SMOVL C00398 BC00398 V=800.0  +MOVJ EC00398
SMOVL C00399 BC00399 V=1000.0  +MOVJ EC00399
SMOVL C00400 BC00400 V=1000.0  +MOVJ EC00400
SFTOF3D
'EndPath W3863
MOVJ C00401 BC00401 VJ=100.00  +MOVJ EC00401 VJ=100.00
MOVJ C00402 BC00402 VJ=100.00  +MOVJ EC00402 VJ=100.00
'Path W3864
SFTOF3D
SFTON3D P033
MOVJ C00403 BC00403 VJ=100.00  +MOVJ EC00403 VJ=100.00
SMOVL C00404 BC00404 V=800.0  +MOVJ EC00404
SMOVL C00405 BC00405 V=166.7 PL=0  +MOVJ EC00405
ARCON
SMOVL C00406 BC00406 V=10.0  +MOVJ EC00406
SFTON3D P034
SMOVL C00407 BC00407 V=10.0  +MOVJ EC00407
SMOVL C00408 BC00408 V=10.0  +MOVJ EC00408
ARCOF
SMOVL C00409 BC00409 V=800.0  +MOVJ EC00409
SMOVL C00410 BC00410 V=1000.0  +MOVJ EC00410
SMOVL C00411 BC00411 V=1000.0  +MOVJ EC00411
SFTOF3D
'EndPath W3864
MOVJ C00412 BC00412 VJ=100.00  +MOVJ EC00412 VJ=100.00
'Path W3865
SFTOF3D
SFTON3D P032
MOVJ C00413 BC00413 VJ=100.00  +MOVJ EC00413 VJ=100.00
MOVJ C00414 BC00414 VJ=100.00  +MOVJ EC00414 VJ=100.00
SMOVL C00415 BC00415 V=800.0  +MOVJ EC00415
SMOVL C00416 BC00416 V=166.7 PL=0  +MOVJ EC00416
ARCON
SMOVL C00417 BC00417 V=9.2  +MOVJ EC00417
SFTON3D P031
SMOVL C00418 BC00418 V=9.2  +MOVJ EC00418
SMOVL C00419 BC00419 V=9.2  +MOVJ EC00419
ARCOF
SMOVL C00420 BC00420 V=800.0  +MOVJ EC00420
SMOVL C00421 BC00421 V=1000.0  +MOVJ EC00421
SFTOF3D
'EndPath W3865
MOVJ C00422 BC00422 VJ=100.00  +MOVJ EC00422 VJ=100.00
'Down
MOVJ C00423 BC00423 VJ=100.00  +MOVJ EC00423 VJ=100.00
MOVJ C00424 BC00424 VJ=100.00  +MOVJ EC00424 VJ=100.00
'Path W3867
SFTOF3D
SFTON3D P026
MOVJ C00425 BC00425 VJ=100.00  +MOVJ EC00425 VJ=100.00
SMOVL C00426 BC00426 V=800.0  +MOVJ EC00426
SMOVL C00427 BC00427 V=150.0 PL=0  +MOVJ EC00427
MACRO1 MJ#(0) ARGF22
ARCON
SMOVC C00428 BC00428 V=9.5  +MOVJ EC00428
SMOVC C00429 BC00429 V=9.5  +MOVJ EC00429
SFTON3D P025
SMOVC C00430 BC00430 V=9.5  +MOVJ EC00430
SMOVL C00431 BC00431 V=9.5  +MOVJ EC00431
ARCOF
SMOVL C00432 BC00432 V=800.0  +MOVJ EC00432
SMOVL C00433 BC00433 V=1000.0  +MOVJ EC00433
SFTOF3D
'EndPath W3867
MOVJ C00434 BC00434 VJ=100.00  +MOVJ EC00434 VJ=100.00
MOVJ C00435 BC00435 VJ=100.00  +MOVJ EC00435 VJ=100.00
MOVJ C00436 BC00436 VJ=100.00  +MOVJ EC00436 VJ=100.00
'Path W3868
SFTOF3D
SFTON3D P022
MOVJ C00437 BC00437 VJ=100.00  +MOVJ EC00437 VJ=100.00
MOVJ C00438 BC00438 VJ=100.00  +MOVJ EC00438 VJ=100.00
SMOVL C00439 BC00439 V=800.0  +MOVJ EC00439
SMOVL C00440 BC00440 V=166.7 PL=0  +MOVJ EC00440
MACRO1 MJ#(0) ARGF9
ARCON
SMOVL C00441 BC00441 V=10.0  +MOVJ EC00441
SMOVL C00442 BC00442 V=10.0  +MOVJ EC00442
SMOVL C00443 BC00443 V=10.0  +MOVJ EC00443
SMOVL C00444 BC00444 V=10.0  +MOVJ EC00444
SMOVL C00445 BC00445 V=10.0  +MOVJ EC00445
SMOVL C00446 BC00446 V=10.0  +MOVJ EC00446
SMOVL C00447 BC00447 V=10.0  +MOVJ EC00447
SMOVL C00448 BC00448 V=10.0  +MOVJ EC00448
SMOVL C00449 BC00449 V=10.0  +MOVJ EC00449
ARCOF
SMOVL C00450 BC00450 V=800.0  +MOVJ EC00450
SMOVL C00451 BC00451 V=1000.0  +MOVJ EC00451
SFTOF3D
'EndPath W3868
MOVJ C00452 BC00452 VJ=100.00  +MOVJ EC00452 VJ=100.00
SFTOF3D
'EndPath W3869
MOVJ C00453 BC00453 VJ=100.00  +MOVJ EC00453 VJ=100.00
'Path W3896
SFTOF3D
SFTON3D P020
MOVJ C00454 BC00454 VJ=100.00  +MOVJ EC00454 VJ=100.00
SMOVL C00455 BC00455 V=800.0  +MOVJ EC00455
SMOVL C00456 BC00456 V=150.0 PL=0  +MOVJ EC00456
ARCON
SMOVL C00457 BC00457 V=10.0  +MOVJ EC00457
ARCOF
SMOVL C00458 BC00458 V=800.0  +MOVJ EC00458
SFTOF3D
'EndPath W3896
MOVJ C00459 BC00459 VJ=100.00  +MOVJ EC00459 VJ=100.00
MOVJ C00460 BC00460 VJ=100.00  +MOVJ EC00460 VJ=100.00
MOVJ C00461 BC00461 VJ=100.00  +MOVJ EC00461 VJ=100.00
'Path W3866
SFTOF3D
SFTON3D P023
MOVJ C00462 BC00462 VJ=100.00  +MOVJ EC00462 VJ=100.00
SMOVL C00463 BC00463 V=800.0  +MOVJ EC00463
SMOVC C00464 BC00464 V=150.0 PL=0  +MOVJ EC00464
MACRO1 MJ#(0) ARGF22
ARCON
SWVON WEV#(108)
SMOVC C00465 BC00465 V=9.5  +MOVJ EC00465
SMOVC C00466 BC00466 V=9.5  +MOVJ EC00466
SFTON3D P024
SMOVC C00467 BC00467 V=9.5  +MOVJ EC00467
SMOVC C00468 BC00468 V=9.5  +MOVJ EC00468
SMOVC C00469 BC00469 V=9.5  +MOVJ EC00469
ARCOF
SWVOF
SMOVL C00470 BC00470 V=800.0  +MOVJ EC00470
SMOVL C00471 BC00471 V=1000.0  +MOVJ EC00471
SFTOF3D
'EndPath W3866
MOVJ C00472 BC00472 VJ=100.00  +MOVJ EC00472 VJ=100.00
MOVJ C00473 BC00473 VJ=100.00  +MOVJ EC00473 VJ=100.00
SFTOF3D
MOVJ C00474 BC00474 VJ=100.00  +MOVJ EC00474 VJ=100.00
SMOVL C00475 BC00475 V=800.0  +MOVJ EC00475
MOVJ C00476 BC00476 VJ=100.00  +MOVJ EC00476 VJ=100.00
SFTON3D P056
MOVJ C00477 BC00477 VJ=100.00  +MOVJ EC00477 VJ=100.00
SMOVL C00478 BC00478 V=150.0 PL=0  +MOVJ EC00478
MACRO1 MJ#(0) ARGF9
ARCON
SFTON3D P057
SMOVL C00479 BC00479 V=10.0  +MOVJ EC00479
SMOVC C00480 BC00480 V=13.3  +MOVJ EC00480
SMOVC C00481 BC00481 V=13.3  +MOVJ EC00481
SMOVC C00482 BC00482 V=13.3  +MOVJ EC00482
SFTON3D P056
SMOVL C00483 BC00483 V=10.0  +MOVJ EC00483
SMOVL C00484 BC00484 V=10.0  +MOVJ EC00484
SMOVC C00485 BC00485 V=13.3  +MOVJ EC00485
SMOVC C00486 BC00486 V=13.3  +MOVJ EC00486
SMOVC C00487 BC00487 V=13.3  +MOVJ EC00487
ARCOF
SMOVL C00488 BC00488 V=166.7  +MOVJ EC00488
SFTOF3D
SMOVL C00489 BC00489 V=666.7  +MOVJ EC00489
SMOVL C00490 BC00490 V=666.7  +MOVJ EC00490
SFTON3D P054
SMOVL C00491 BC00491 V=150.0 PL=0  +MOVJ EC00491
MACRO1 MJ#(0) ARGF9
ARCON
SFTON3D P055
SMOVL C00492 BC00492 V=10.0  +MOVJ EC00492
SMOVC C00493 BC00493 V=13.3  +MOVJ EC00493
SMOVC C00494 BC00494 V=13.3  +MOVJ EC00494
SMOVC C00495 BC00495 V=13.3  +MOVJ EC00495
SFTON3D P054
SMOVL C00496 BC00496 V=10.0  +MOVJ EC00496
SMOVL C00497 BC00497 V=10.0  +MOVJ EC00497
SMOVC C00498 BC00498 V=13.3  +MOVJ EC00498
SMOVC C00499 BC00499 V=13.3  +MOVJ EC00499
SMOVC C00500 BC00500 V=13.3  +MOVJ EC00500
ARCOF
SMOVL C00501 BC00501 V=166.7  +MOVJ EC00501
SFTOF3D
MOVL C00502 BC00502 V=666.7  +MOVJ EC00502 VJ=0.78
MOVL C00503 BC00503 V=666.7  +MOVJ EC00503 VJ=0.78
MOVL C00504 BC00504 V=666.7  +MOVJ EC00504 VJ=0.78
MOVJ C00505 BC00505 VJ=100.00  +MOVJ EC00505 VJ=0.78
SFTON3D P060
SMOVL C00506 BC00506 V=150.0 PL=0  +MOVJ EC00506
MACRO1 MJ#(0) ARGF9
ARCON
SFTON3D P061
SMOVL C00507 BC00507 V=10.0  +MOVJ EC00507
SMOVC C00508 BC00508 V=15.0  +MOVJ EC00508
SMOVC C00509 BC00509 V=15.0  +MOVJ EC00509
SMOVC C00510 BC00510 V=13.3  +MOVJ EC00510
SFTON3D P060
SMOVL C00511 BC00511 V=10.0  +MOVJ EC00511
SMOVL C00512 BC00512 V=10.0  +MOVJ EC00512
SMOVC C00513 BC00513 V=13.3  +MOVJ EC00513
SMOVC C00514 BC00514 V=13.3  +MOVJ EC00514
SMOVC C00515 BC00515 V=15.0  +MOVJ EC00515
ARCOF
SMOVL C00516 BC00516 V=166.7  +MOVJ EC00516
SFTOF3D
MOVJ C00517 BC00517 VJ=100.00  +MOVJ EC00517 VJ=100.00
MOVJ C00518 BC00518 VJ=100.00  +MOVJ EC00518 VJ=100.00
SFTON3D P059
SMOVL C00519 BC00519 V=150.0 PL=0  +MOVJ EC00519
MACRO1 MJ#(0) ARGF9
ARCON
SFTON3D P058
SMOVL C00520 BC00520 V=10.0  +MOVJ EC00520
SMOVC C00521 BC00521 V=13.3  +MOVJ EC00521
SMOVC C00522 BC00522 V=13.3  +MOVJ EC00522
SMOVC C00523 BC00523 V=13.3  +MOVJ EC00523
SFTON3D P059
SMOVL C00524 BC00524 V=10.0  +MOVJ EC00524
SMOVL C00525 BC00525 V=10.0  +MOVJ EC00525
SMOVC C00526 BC00526 V=13.3  +MOVJ EC00526
SMOVC C00527 BC00527 V=13.3  +MOVJ EC00527
SMOVC C00528 BC00528 V=13.3  +MOVJ EC00528
ARCOF
SMOVL C00529 BC00529 V=166.7  +MOVJ EC00529
SFTOF3D
MOVJ C00530 BC00530 VJ=100.00  +MOVJ EC00530 VJ=100.00
MOVJ C00531 BC00531 VJ=100.00  +MOVJ EC00531 VJ=100.00
SFTON3D P063
SMOVL C00532 BC00532 V=150.0 PL=0  +MOVJ EC00532
MACRO1 MJ#(0) ARGF9
ARCON
SFTON3D P062
SMOVL C00533 BC00533 V=10.0  +MOVJ EC00533
SMOVC C00534 BC00534 V=13.3  +MOVJ EC00534
SMOVC C00535 BC00535 V=13.3  +MOVJ EC00535
SMOVC C00536 BC00536 V=13.3  +MOVJ EC00536
SFTON3D P063
SMOVL C00537 BC00537 V=10.0  +MOVJ EC00537
SMOVL C00538 BC00538 V=10.0  +MOVJ EC00538
SMOVC C00539 BC00539 V=13.3  +MOVJ EC00539
SMOVC C00540 BC00540 V=13.3  +MOVJ EC00540
SMOVC C00541 BC00541 V=13.3  +MOVJ EC00541
ARCOF
SMOVL C00542 BC00542 V=166.7  +MOVJ EC00542
SFTOF3D
MOVJ C00543 BC00543 VJ=100.00  +MOVJ EC00543 VJ=100.00
MOVJ C00544 BC00544 VJ=100.00  +MOVJ EC00544 VJ=100.00
SFTON3D P072
SMOVL C00545 BC00545 V=150.0 PL=0  +MOVJ EC00545
MACRO1 MJ#(0) ARGF9
ARCON
SFTON3D P071
SMOVL C00546 BC00546 V=10.0  +MOVJ EC00546
SMOVC C00547 BC00547 V=13.3  +MOVJ EC00547
SMOVC C00548 BC00548 V=13.3  +MOVJ EC00548
SMOVC C00549 BC00549 V=13.3  +MOVJ EC00549
SMOVL C00550 BC00550 V=10.0  +MOVJ EC00550
SFTON3D P070
SMOVL C00551 BC00551 V=10.0  +MOVJ EC00551
SMOVL C00552 BC00552 V=10.0  +MOVJ EC00552
ARCOF
SMOVL C00553 BC00553 V=166.7  +MOVJ EC00553
SFTOF3D
MOVJ C00554 BC00554 VJ=100.00  +MOVJ EC00554 VJ=100.00
MOVJ C00555 BC00555 VJ=100.00  +MOVJ EC00555 VJ=100.00
SFTON3D P065
SMOVL C00556 BC00556 V=150.0 PL=0  +MOVJ EC00556
MACRO1 MJ#(0) ARGF9
ARCON
SFTON3D P064
SMOVL C00557 BC00557 V=10.0  +MOVJ EC00557
SMOVC C00558 BC00558 V=13.3  +MOVJ EC00558
SMOVC C00559 BC00559 V=13.3  +MOVJ EC00559
SMOVC C00560 BC00560 V=13.3  +MOVJ EC00560
SFTON3D P065
SMOVL C00561 BC00561 V=10.0  +MOVJ EC00561
SMOVL C00562 BC00562 V=10.0  +MOVJ EC00562
SMOVC C00563 BC00563 V=13.3  +MOVJ EC00563
SMOVC C00564 BC00564 V=13.3  +MOVJ EC00564
SMOVC C00565 BC00565 V=13.3  +MOVJ EC00565
ARCOF
SMOVL C00566 BC00566 V=166.7  +MOVJ EC00566
SFTOF3D
MOVJ C00567 BC00567 VJ=100.00  +MOVJ EC00567 VJ=100.00
MOVJ C00568 BC00568 VJ=100.00  +MOVJ EC00568 VJ=100.00
MOVJ C00569 BC00569 VJ=100.00  +MOVJ EC00569 VJ=100.00
SFTON3D P051
SMOVL C00570 BC00570 V=150.0 PL=0  +MOVJ EC00570
MACRO1 MJ#(0) ARGF9
ARCON
SMOVL C00571 BC00571 V=10.8  +MOVJ EC00571
SMOVC C00572 BC00572 V=13.3  +MOVJ EC00572
SMOVC C00573 BC00573 V=13.3  +MOVJ EC00573
SMOVC C00574 BC00574 V=13.3  +MOVJ EC00574
SFTON3D P052
SMOVL C00575 BC00575 V=11.7  +MOVJ EC00575
SFTON3D P053
SMOVL C00576 BC00576 V=11.7  +MOVJ EC00576
SMOVC C00577 BC00577 V=13.3  +MOVJ EC00577
SMOVC C00578 BC00578 V=13.3  +MOVJ EC00578
SMOVC C00579 BC00579 V=13.3  +MOVJ EC00579
ARCOF
SMOVL C00580 BC00580 V=166.7  +MOVJ EC00580
SFTOF3D
MOVL C00581 BC00581 V=1000.0  +MOVJ EC00581 VJ=100.00
MOVJ C00582 BC00582 VJ=100.00  +MOVJ EC00582 VJ=100.00
CALL JOB:CLEAN-R1_KM_3P
MOVJ C00583 BC00583 VJ=100.00  +MOVJ EC00583 VJ=0.78
MOVJ C00584 BC00584 VJ=100.00  +MOVJ EC00584 VJ=100.00
MOVJ C00585 BC00585 VJ=100.00  +MOVJ EC00585 VJ=100.00
MOVJ C00586 BC00586 VJ=100.00  +MOVJ EC00586 VJ=100.00
MOVJ C00587 BC00587 VJ=100.00  +MOVJ EC00587 VJ=100.00
MOVJ C00588 BC00588 VJ=100.00  +MOVJ EC00588 VJ=100.00
MOVJ C00589 BC00589 VJ=100.00  +MOVJ EC00589 VJ=100.00
MOVJ C00590 BC00590 VJ=100.00  +MOVJ EC00590 VJ=100.00
MOVJ C00591 BC00591 VJ=100.00  +MOVJ EC00591 VJ=100.00
MOVJ C00592 BC00592 VJ=100.00  +MOVJ EC00592 VJ=100.00
SMOVL C00593 BC00593 V=333.3  +MOVJ EC00593
SMOVL C00594 BC00594 V=333.3  +MOVJ EC00594
MOVJ C00595 BC00595 VJ=100.00  +MOVJ EC00595 VJ=100.00
SMOVL C00596 BC00596 V=333.3  +MOVJ EC00596
SMOVL C00597 BC00597 V=166.7  +MOVJ EC00597
SREFP 3 C00598 BC00598  +REFP EC00598
CALL JOB:SEARCH-R1-S13D
SET P051 P006
SFTON3D P051
SMOVL C00599 BC00599 V=166.7  +MOVJ EC00599
SREFP 3 C00600 BC00600  +REFP EC00600
CALL JOB:SEARCH-R1-S13D
SET P051 P006
SFTON3D P051
SMOVL C00601 BC00601 V=166.7  +MOVJ EC00601
SREFP 3 C00602 BC00602  +REFP EC00602
CALL JOB:SEARCH-R1-S13D
SET P051 P006
SFTON3D P051
SMOVL C00603 BC00603 V=166.7  +MOVJ EC00603
SMOVL C00604 BC00604 V=166.7 PL=0  +MOVJ EC00604
SMOVL C00605 BC00605 V=166.7  +MOVJ EC00605
SREFP 3 C00606 BC00606  +REFP EC00606
CALL JOB:SEARCH-R1-S13D
SET P052 P006
SFTON3D P052
SMOVL C00607 BC00607 V=166.7  +MOVJ EC00607
SREFP 3 C00608 BC00608  +REFP EC00608
CALL JOB:SEARCH-R1-S13D
SET P052 P006
SFTON3D P052
SMOVL C00609 BC00609 V=166.7  +MOVJ EC00609
SMOVL C00610 BC00610 V=333.3 PL=0  +MOVJ EC00610
SMOVL C00611 BC00611 V=166.7  +MOVJ EC00611
SREFP 3 C00612 BC00612  +REFP EC00612
CALL JOB:SEARCH-R1-S13D
SET P053 P006
SFTON3D P053
SMOVL C00613 BC00613 V=166.7  +MOVJ EC00613
SREFP 3 C00614 BC00614  +REFP EC00614
CALL JOB:SEARCH-R1-S13D
SET P053 P006
SFTON3D P053
SMOVL C00615 BC00615 V=166.7  +MOVJ EC00615
SFTOF3D
SFTOF
SFTON3D P051
SMOVL C00616 BC00616 V=333.3  +MOVJ EC00616
SMOVL C00617 BC00617 V=166.7  +MOVJ EC00617
SREFP 3 C00618 BC00618  +REFP EC00618
CALL JOB:SEARCH-R1-S13D
SET P050 P006
SFTON3D P050
SMOVL C00619 BC00619 V=166.7  +MOVJ EC00619
SREFP 3 C00620 BC00620  +REFP EC00620
CALL JOB:SEARCH-R1-S13D
SET P050 P006
SFTON3D P050
SMOVL C00621 BC00621 V=166.7  +MOVJ EC00621
SMOVL C00622 BC00622 V=166.7  +MOVJ EC00622
SREFP 3 C00623 BC00623  +REFP EC00623
CALL JOB:SEARCH-R1-S13D
SET P050 P006
SFTON3D P050
SMOVL C00624 BC00624 V=166.7  +MOVJ EC00624
SFTOF3D
SMOVL C00625 BC00625 V=333.3  +MOVJ EC00625
SMOVL C00626 BC00626 V=166.7  +MOVJ EC00626
SREFP 3 C00627 BC00627  +REFP EC00627
CALL JOB:SEARCH-R1-S13D
SET P054 P006
SFTON3D P054
SMOVL C00628 BC00628 V=166.7  +MOVJ EC00628
SREFP 3 C00629 BC00629  +REFP EC00629
CALL JOB:SEARCH-R1-S13D
SET P054 P006
SFTON3D P054
SMOVL C00630 BC00630 V=166.7  +MOVJ EC00630
SMOVL C00631 BC00631 V=166.7  +MOVJ EC00631
SREFP 3 C00632 BC00632  +REFP EC00632
CALL JOB:SEARCH-R1-S13D
SET P054 P006
SFTON3D P054
SMOVL C00633 BC00633 V=166.7  +MOVJ EC00633
SMOVL C00634 BC00634 V=333.3  +MOVJ EC00634
SMOVL C00635 BC00635 V=166.7  +MOVJ EC00635
SREFP 3 C00636 BC00636  +REFP EC00636
CALL JOB:SEARCH-R1-S13D
SET P055 P006
SFTON3D P055
SMOVL C00637 BC00637 V=166.7  +MOVJ EC00637
SREFP 3 C00638 BC00638  +REFP EC00638
CALL JOB:SEARCH-R1-S13D
SET P055 P006
SFTON3D P055
SMOVL C00639 BC00639 V=166.7  +MOVJ EC00639
SREFP 3 C00640 BC00640  +REFP EC00640
CALL JOB:SEARCH-R1-S13D
SET P055 P006
SFTON3D P055
SMOVL C00641 BC00641 V=166.7  +MOVJ EC00641
MOVJ C00642 BC00642 VJ=100.00  +MOVJ EC00642 VJ=100.00
MOVL C00643 BC00643 V=333.3  +MOVJ EC00643 VJ=100.00
SMOVL C00644 BC00644 V=166.7  +MOVJ EC00644
SREFP 3 C00645 BC00645  +REFP EC00645
CALL JOB:SEARCH-R1-S13D
SET P056 P006
SFTON3D P056
SMOVL C00646 BC00646 V=166.7  +MOVJ EC00646
SREFP 3 C00647 BC00647  +REFP EC00647
CALL JOB:SEARCH-R1-S13D
SET P056 P006
SFTON3D P056
SMOVL C00648 BC00648 V=166.7  +MOVJ EC00648
SMOVL C00649 BC00649 V=333.3  +MOVJ EC00649
SMOVL C00650 BC00650 V=166.7  +MOVJ EC00650
SREFP 3 C00651 BC00651  +REFP EC00651
CALL JOB:SEARCH-R1-S13D
SET P057 P006
SFTON3D P057
SMOVL C00652 BC00652 V=166.7  +MOVJ EC00652
SREFP 3 C00653 BC00653  +REFP EC00653
CALL JOB:SEARCH-R1-S13D
SET P057 P006
SFTON3D P057
SMOVL C00654 BC00654 V=166.7  +MOVJ EC00654
SMOVL C00655 BC00655 V=333.3  +MOVJ EC00655
SMOVL C00656 BC00656 V=166.7  +MOVJ EC00656
SREFP 3 C00657 BC00657  +REFP EC00657
CALL JOB:SEARCH-R1-S13D
SET P058 P006
SFTON3D P058
SMOVL C00658 BC00658 V=166.7  +MOVJ EC00658
SREFP 3 C00659 BC00659  +REFP EC00659
CALL JOB:SEARCH-R1-S13D
SET P058 P006
SFTON3D P058
SMOVL C00660 BC00660 V=166.7  +MOVJ EC00660
SFTOF3D
MOVL C00661 BC00661 V=333.3  +MOVJ EC00661 VJ=100.00
MOVL C00662 BC00662 V=333.3  +MOVJ EC00662 VJ=100.00
SMOVL C00663 BC00663 V=166.7  +MOVJ EC00663
SREFP 3 C00664 BC00664  +REFP EC00664
CALL JOB:SEARCH-R1-S13D
SET P059 P006
SFTON3D P059
SMOVL C00665 BC00665 V=166.7  +MOVJ EC00665
SREFP 3 C00666 BC00666  +REFP EC00666
CALL JOB:SEARCH-R1-S13D
SET P059 P006
SFTON3D P059
SMOVL C00667 BC00667 V=166.7  +MOVJ EC00667
SREFP 3 C00668 BC00668  +REFP EC00668
CALL JOB:SEARCH-R1-S13D
SET P059 P006
SFTON3D P059
SMOVL C00669 BC00669 V=166.7  +MOVJ EC00669
MOVL C00670 BC00670 V=333.3  +MOVJ EC00670 VJ=100.00
SMOVL C00671 BC00671 V=166.7  +MOVJ EC00671
SREFP 3 C00672 BC00672  +REFP EC00672
CALL JOB:SEARCH-R1-S13D
SET P060 P006
SFTON3D P060
SMOVL C00673 BC00673 V=166.7  +MOVJ EC00673
SREFP 3 C00674 BC00674  +REFP EC00674
CALL JOB:SEARCH-R1-S13D
SET P060 P006
SFTON3D P060
SMOVL C00675 BC00675 V=166.7  +MOVJ EC00675
SREFP 3 C00676 BC00676  +REFP EC00676
CALL JOB:SEARCH-R1-S13D
SET P060 P006
SFTON3D P060
SMOVL C00677 BC00677 V=166.7  +MOVJ EC00677
SFTOF3D
SFTON3D P060
MACRO1 MJ#(0) ARGF9
SMOVL C00678 BC00678 V=150.0 PL=0  +MOVJ EC00678
ARCON
SMOVL C00679 BC00679 V=10.0  +MOVJ EC00679
SMOVC C00680 BC00680 V=13.3  +MOVJ EC00680
SMOVC C00681 BC00681 V=13.3  +MOVJ EC00681
SMOVC C00682 BC00682 V=13.3  +MOVJ EC00682
SFTON3D P059
SMOVL C00683 BC00683 V=10.0  +MOVJ EC00683
SMOVL C00684 BC00684 V=10.0  +MOVJ EC00684
SMOVC C00685 BC00685 V=13.3  +MOVJ EC00685
SMOVC C00686 BC00686 V=13.3  +MOVJ EC00686
SMOVC C00687 BC00687 V=13.3  +MOVJ EC00687
SFTON3D P060
SMOVL C00688 BC00688 V=10.0  +MOVJ EC00688
ARCOF
SMOVL C00689 BC00689 V=166.7  +MOVJ EC00689
SFTOF3D
MOVL C00690 BC00690 V=333.3  +MOVJ EC00690 VJ=100.00
MOVL C00691 BC00691 V=333.3  +MOVJ EC00691 VJ=100.00
MOVL C00692 BC00692 V=333.3  +MOVJ EC00692 VJ=100.00
SFTON3D P056
MOVL C00693 BC00693 V=333.3  +MOVJ EC00693 VJ=100.00
SMOVL C00694 BC00694 V=150.0 PL=0  +MOVJ EC00694
ARCON
SMOVL C00695 BC00695 V=10.0  +MOVJ EC00695
SMOVC C00696 BC00696 V=13.3  +MOVJ EC00696
SMOVC C00697 BC00697 V=13.3  +MOVJ EC00697
SMOVC C00698 BC00698 V=13.3  +MOVJ EC00698
SMOVL C00699 BC00699 V=10.0  +MOVJ EC00699
SFTON3D P057
SMOVL C00700 BC00700 V=10.0  +MOVJ EC00700
SMOVC C00701 BC00701 V=13.3  +MOVJ EC00701
SFTON3D P058
SMOVC C00702 BC00702 V=13.3  +MOVJ EC00702
SMOVC C00703 BC00703 V=13.3  +MOVJ EC00703
SMOVL C00704 BC00704 V=10.0  +MOVJ EC00704
ARCOF
SMOVL C00705 BC00705 V=166.7  +MOVJ EC00705
SFTOF3D
MOVL C00706 BC00706 V=333.3  +MOVJ EC00706 VJ=100.00
MOVJ C00707 BC00707 VJ=100.00  +MOVJ EC00707 VJ=100.00
MOVJ C00708 BC00708 VJ=100.00  +MOVJ EC00708 VJ=100.00
SFTON3D P054
MACRO1 MJ#(0) ARGF9
SMOVL C00709 BC00709 V=150.0 PL=0  +MOVJ EC00709
ARCON
SFTON3D P055
SMOVL C00710 BC00710 V=10.0  +MOVJ EC00710
SMOVC C00711 BC00711 V=13.3  +MOVJ EC00711
SMOVC C00712 BC00712 V=13.3  +MOVJ EC00712
SMOVC C00713 BC00713 V=13.3  +MOVJ EC00713
SFTON3D P054
SMOVL C00714 BC00714 V=10.0  +MOVJ EC00714
SMOVL C00715 BC00715 V=10.0  +MOVJ EC00715
SMOVC C00716 BC00716 V=13.3  +MOVJ EC00716
SMOVC C00717 BC00717 V=13.3  +MOVJ EC00717
SMOVC C00718 BC00718 V=13.3  +MOVJ EC00718
ARCOF
SMOVL C00719 BC00719 V=166.7  +MOVJ EC00719
SFTOF3D
MOVJ C00720 BC00720 VJ=50.00  +MOVJ EC00720 VJ=100.00
MOVJ C00721 BC00721 VJ=50.00  +MOVJ EC00721 VJ=50.00
SFTON3D P051
MACRO1 MJ#(0) ARGF9
SMOVL C00722 BC00722 V=150.0 PL=0  +MOVJ EC00722
ARCON
SFTON3D P050
SMOVL C00723 BC00723 V=10.0  +MOVJ EC00723
SMOVC C00724 BC00724 V=13.3  +MOVJ EC00724
SMOVC C00725 BC00725 V=13.3  +MOVJ EC00725
SMOVC C00726 BC00726 V=13.3  +MOVJ EC00726
SFTON3D P051
SMOVL C00727 BC00727 V=10.0  +MOVJ EC00727
SMOVL C00728 BC00728 V=10.0  +MOVJ EC00728
SMOVC C00729 BC00729 V=13.3  +MOVJ EC00729
SMOVC C00730 BC00730 V=13.3  +MOVJ EC00730
SMOVC C00731 BC00731 V=13.3  +MOVJ EC00731
ARCOF
SMOVL C00732 BC00732 V=166.7  +MOVJ EC00732
SFTOF3D
MOVJ C00733 BC00733 VJ=50.00  +MOVJ EC00733 VJ=50.00
SFTON3D P052
SMOVL C00734 BC00734 V=150.0 PL=0  +MOVJ EC00734
ARCON
SWVON WEV#(70)
SMOVL C00735 BC00735 V=6.7  +MOVJ EC00735
ARCOF
SWVOF
SMOVL C00736 BC00736 V=166.7  +MOVJ EC00736
SMOVL C00737 BC00737 V=166.7  +MOVJ EC00737
SMOVL C00738 BC00738 V=150.0 PL=0  +MOVJ EC00738
ARCON
SWVON WEV#(70)
SMOVL C00739 BC00739 V=6.7  +MOVJ EC00739
SFTON3D P053
SMOVL C00740 BC00740 V=6.7  +MOVJ EC00740
ARCOF
SWVOF
SMOVL C00741 BC00741 V=166.7  +MOVJ EC00741
SMOVL C00742 BC00742 V=166.7  +MOVJ EC00742
SMOVL C00743 BC00743 V=150.0 PL=0  +MOVJ EC00743
ARCON
SWVON WEV#(70)
SMOVL C00744 BC00744 V=6.7  +MOVJ EC00744
ARCOF
SWVOF
SMOVL C00745 BC00745 V=166.7  +MOVJ EC00745
SFTOF3D
SMOVL C00746 BC00746 V=666.7  +MOVJ EC00746
SMOVL C00747 BC00747 V=666.7  +MOVJ EC00747
MOVL C00748 BC00748 V=1000.0  +MOVJ EC00748 VJ=50.00
MOVJ C00749 BC00749 VJ=100.00  +MOVJ EC00749 VJ=50.00
MOVJ C00750 BC00750 VJ=100.00  +MOVJ EC00750 VJ=100.00
'
END
